// TIA Portal V16 export
// export: Created 2021-04-12T08:07:25.9683963Z, ExportSetting WithDefaults, DisplayName Totally Integrated Automation Portal, DisplayVersion V16, DisplayName TIA Portal Version Control Interface, DisplayVersion V16, DisplayName TIA Portal Openness, DisplayVersion V16, DisplayName STEP 7 Professional, DisplayVersion V16, DisplayName STEP 7 Safety, DisplayVersion V16, DisplayName WinCC Unified SCADA Engineering System, DisplayVersion V16
FUNCTION_BLOCK "AutoMode"   // FB20, LAD
TITLE = Автоматический режим
{ S7_Optimized_Access := 'TRUE' }
VERSION : 0.1
// //setWeight - уставка веса в упаковке => используется при подсчете уставок в бункера
// //speed_inConveyer - уставка скорости на питателе в %
// //speedVibro - уставка скорости вибрации в %
// //maxWeightBunker - максимальный вес в один бункер => используется при подсчете уставок в бункера
// //workPlavnik - использовать ли плавник во время работы 
// //measurementError - допустимая погрешность на итоговый вес => используется при поиске подходящих бункеров при сбросе
// //mediumWeightProduct - средний вес продукта => используется при подсчете уставок в бункера
// stored: AutoNumber false, IsIECCheckEnabled false, IsRetainMemResEnabled false, MemoryReserve 100, SetENOAutomatically false, UDAEnableTagReadback false
   VAR_IN_OUT
      enableAutoMode : Bool;   // разрешение на переход в автоматический режим
      isFinishPreWork : Bool;   // сигнал об окончании подготовки к автоматическому режиму
      isStartAutoMode : Bool;   // сигнал что автоматический режим запущен
   END_VAR
   VAR
      TaskSetWeight : Real;   // целевой вес который ищем в сортировке
      SetWeightBunker : Array[0..12] of Real;   // уставки весов в бункера
      currentWeightBunker : Array[0..12] of Real;
      readyToSort : Array[0..12] of Bool;   // массив говорящий какие бункера готовы к сортировке
      readyToDrop : Array[0..12] of Bool;   // массив говорящий какие бункера надо сбросить
      readyToDropYP : Array[0..2] of Bool;
      isWorkWithBunker : Array[0..12] of Bool;   // массив разрешающий бункерам работать
      preWorkAutoMode : Struct
         isFinishPreWork : Bool;
         alarmStop : Bool;
      END_STRUCT;
      preWork_AM_FB : "preWork_AM";
      workPackingMachine_AM_FB : "workPackingMachine_AM";
      workInConveyer_AM_FB : "workInConveyer_AM";
      controlFllipper_AM_FB : "controlValve";
      workVibroLot_AM_FB : Array[0..12] of "workVibroLot_AM";
      workVibroTable_AM_FB : "workVibroTable_AM";
      weightModule_AM_FB : "weightModule_AM";
      Sorting_AM_FB : "Sorting_AM";
      setWeightBunker_FB : "setWeightBunker_AM";
      blockSorting : Bool;   // запрет на сортировку в блоке сортировке
      openFlipper : Bool;
      hmiYpDropWeight : Array[0..2] of Real;
      hmiYpDropError : Array[0..2] of Real;
      Sorting_AM_withBuffer_FB { S7_SetPoint := 'True'} : "Sorting_AM_withBuffer";
   END_VAR
   VAR_TEMP
      "!!!!!" : Array[0..1] of Bool;
      i : DInt;
      tmpStableWeightBunker : Array[0..12] of Real;
   END_VAR
BEGIN

REGION Network 1: Аварийный останов
   // По нажатию кнопки Стоп и Аварийный стоп
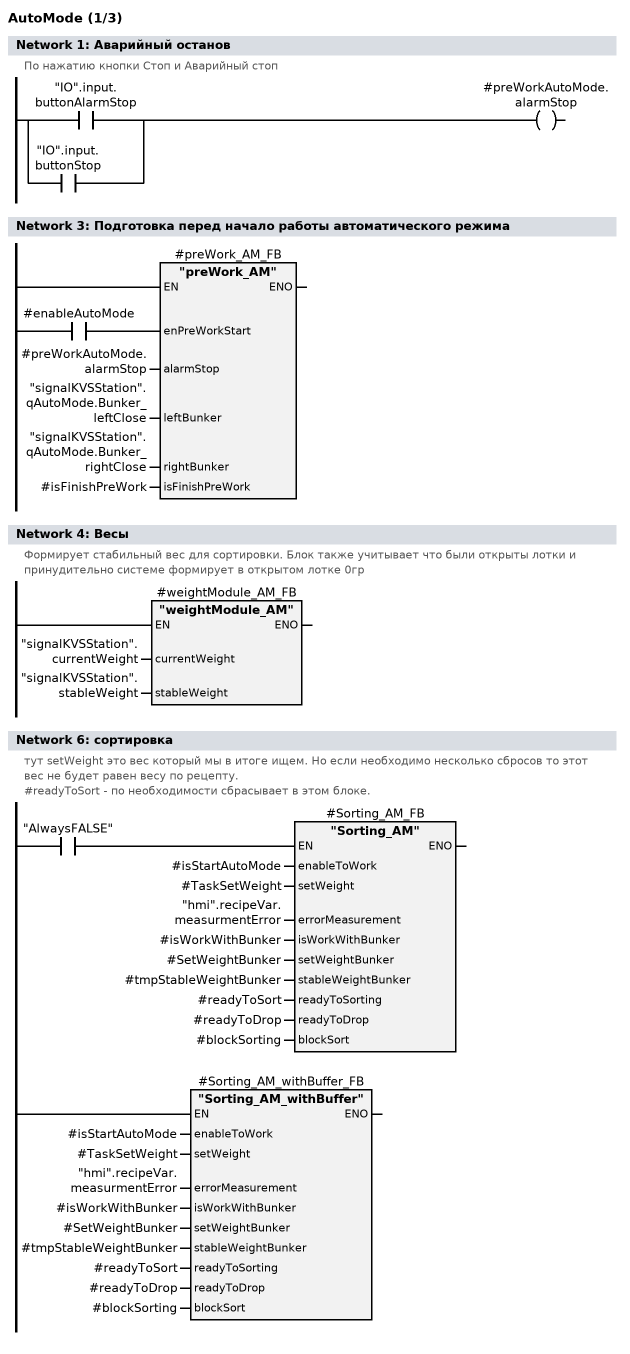
   RUNG wire#powerrail
      Contact( "IO".input.buttonAlarmStop )
      wire#w1
      Coil( #preWorkAutoMode.alarmStop )
   END_RUNG
   RUNG wire#powerrail
      Contact( "IO".input.buttonStop )
   END_RUNG wire#w1
   // the same network as SCL:
   #preWorkAutoMode.alarmStop := "IO".input.buttonAlarmStop OR "IO".input.buttonStop;
END_REGION

REGION Network 2 (SCL): статусы автоматического режима
   IF #enableAutoMode THEN
       IF NOT (#isFinishPreWork) THEN
           "hmi".readySystem := 2;
       ELSE
           IF NOT (#isStartAutoMode) THEN
               "hmi".readySystem := 0;
           ELSE
               "hmi".readySystem := 1;
           END_IF;
       END_IF;
   END_IF;
END_REGION

REGION Network 3: Подготовка перед начало работы автоматического режима
   RUNG wire#powerrail
      #preWork_AM_FB(enPreWorkStart := wire#w1, alarmStop := #preWorkAutoMode.alarmStop, leftBunker := "signalKVSStation".qAutoMode.Bunker_leftClose, rightBunker := "signalKVSStation".qAutoMode.Bunker_rightClose, isFinishPreWork := #isFinishPreWork)
   END_RUNG
   RUNG wire#powerrail
      Contact( #enableAutoMode )
   END_RUNG wire#w1
   // the same network as SCL:
   #preWork_AM_FB(enPreWorkStart := #enableAutoMode,   // "preWork_AM"
                  alarmStop := #preWorkAutoMode.alarmStop,
                  leftBunker := "signalKVSStation".qAutoMode.Bunker_leftClose,
                  rightBunker := "signalKVSStation".qAutoMode.Bunker_rightClose,
                  isFinishPreWork := #isFinishPreWork);
END_REGION

REGION Network 4: Весы
   // Формирует стабильный вес для сортировки. Блок также учитывает что были открыты лотки и принудительно системе формирует в открытом лотке 0гр
   RUNG wire#powerrail
      #weightModule_AM_FB(currentWeight := "signalKVSStation".currentWeight, stableWeight := "signalKVSStation".stableWeight)
   END_RUNG
   // the same network as SCL:
   #weightModule_AM_FB(currentWeight := "signalKVSStation".currentWeight,   // "weightModule_AM"
                       stableWeight := "signalKVSStation".stableWeight);
END_REGION

REGION Network 5 (SCL): выделяем стабильные веса с которыми будем работать
   #i := 0;
   FOR #i := 1 TO 12 DO
       #tmpStableWeightBunker[#i] := "signalKVSStation".stableWeight[#i].weight[0];
       "hmi".weightLine[#i].currentWeightPocket := "signalKVSStation".stableWeight[#i].weight[0];
       "hmi".weightLine[#i].targetWeightPocket := #SetWeightBunker[#i];
   END_FOR;
   #currentWeightBunker := "signalKVSStation".currentWeight;
END_REGION

REGION Network 6: сортировка
   // тут setWeight это вес который мы в итоге ищем. Но если необходимо несколько сбросов то этот вес не будет равен весу по рецепту.
   // #readyToSort - по необходимости сбрасывает в этом блоке.
   RUNG wire#powerrail
      Contact( "AlwaysFALSE" )
      #Sorting_AM_FB(enableToWork := #isStartAutoMode, setWeight := #TaskSetWeight, errorMeasurement := "hmi".recipeVar.measurmentError, isWorkWithBunker := #isWorkWithBunker, setWeightBunker := #SetWeightBunker, stableWeightBunker := #tmpStableWeightBunker, readyToSorting := #readyToSort, readyToDrop := #readyToDrop, blockSort := #blockSorting)
   END_RUNG
   RUNG wire#powerrail
      #Sorting_AM_withBuffer_FB(enableToWork := #isStartAutoMode, setWeight := #TaskSetWeight, errorMeasurement := "hmi".recipeVar.measurmentError, isWorkWithBunker := #isWorkWithBunker, setWeightBunker := #SetWeightBunker, stableWeightBunker := #tmpStableWeightBunker, readyToSorting := #readyToSort, readyToDrop := #readyToDrop, blockSort := #blockSorting)
   END_RUNG
   // the same network as SCL:
   IF "AlwaysFALSE" THEN
       #Sorting_AM_FB(enableToWork := #isStartAutoMode,   // "Sorting_AM"
                      setWeight := #TaskSetWeight,
                      errorMeasurement := "hmi".recipeVar.measurmentError,
                      isWorkWithBunker := #isWorkWithBunker,
                      setWeightBunker := #SetWeightBunker,
                      stableWeightBunker := #tmpStableWeightBunker,
                      readyToSorting := #readyToSort,
                      readyToDrop := #readyToDrop,
                      blockSort := #blockSorting);
   END_IF;
   #Sorting_AM_withBuffer_FB(enableToWork := #isStartAutoMode,   // "Sorting_AM_withBuffer"
                           setWeight := #TaskSetWeight,
                           errorMeasurement := "hmi".recipeVar.measurmentError,
                           isWorkWithBunker := #isWorkWithBunker,
                           setWeightBunker := #SetWeightBunker,
                           stableWeightBunker := #tmpStableWeightBunker,
                           readyToSorting := #readyToSort,
                           readyToDrop := #readyToDrop,
                           blockSort := #blockSorting);
END_REGION

REGION Network 7 (SCL): Перенос данных для панели
   "hmi".permitOn1Bunk := "hmi".permitOn2Bunk := #readyToDrop;
END_REGION

REGION Network 8: Расчет уставок в бункере
   // Здесь происходит расчет уставок на все бункера в зависимости от: веса уставки, максимального веса в один бункер, среднего веса продукта
   // Также управление конвейерами, упаковочными машинами и бункерами
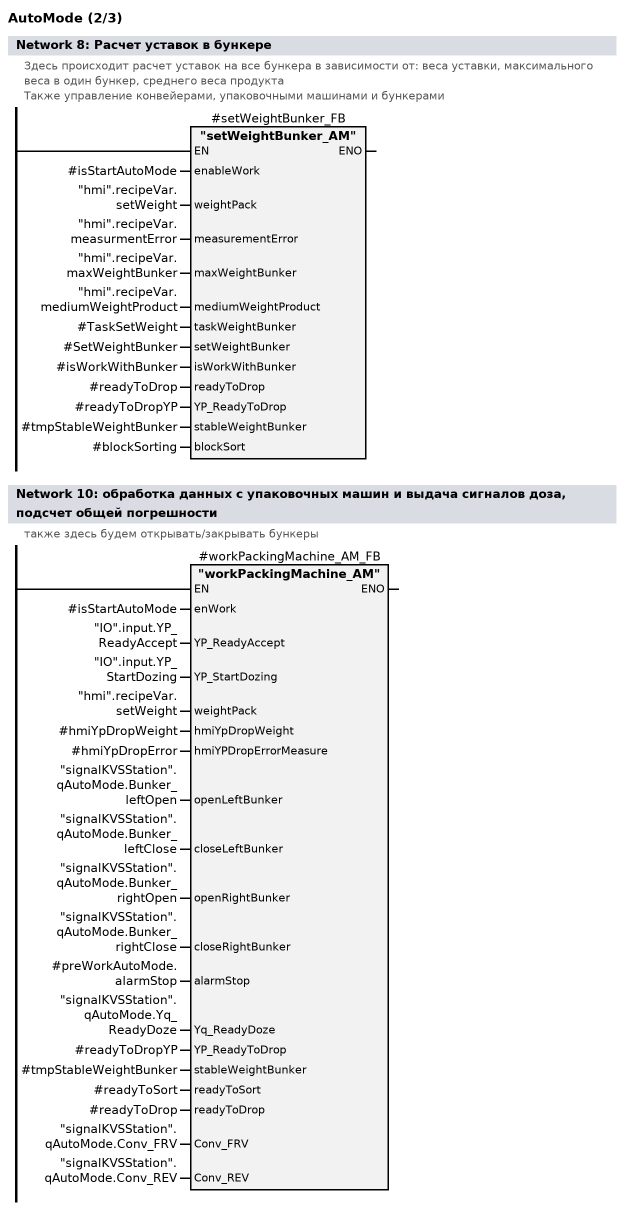
   RUNG wire#powerrail
      #setWeightBunker_FB(enableWork := #isStartAutoMode, weightPack := "hmi".recipeVar.setWeight, measurementError := "hmi".recipeVar.measurmentError, maxWeightBunker := "hmi".recipeVar.maxWeightBunker, mediumWeightProduct := "hmi".recipeVar.mediumWeightProduct, taskWeightBunker := #TaskSetWeight, setWeightBunker := #SetWeightBunker, isWorkWithBunker := #isWorkWithBunker, readyToDrop := #readyToDrop, YP_ReadyToDrop := #readyToDropYP, stableWeightBunker := #tmpStableWeightBunker, blockSort := #blockSorting)
   END_RUNG
   // the same network as SCL:
   #setWeightBunker_FB(enableWork := #isStartAutoMode,   // "setWeightBunker_AM"
                       weightPack := "hmi".recipeVar.setWeight,
                       measurementError := "hmi".recipeVar.measurmentError,
                       maxWeightBunker := "hmi".recipeVar.maxWeightBunker,
                       mediumWeightProduct := "hmi".recipeVar.mediumWeightProduct,
                       taskWeightBunker := #TaskSetWeight,
                       setWeightBunker := #SetWeightBunker,
                       isWorkWithBunker := #isWorkWithBunker,
                       readyToDrop := #readyToDrop,
                       YP_ReadyToDrop := #readyToDropYP,
                       stableWeightBunker := #tmpStableWeightBunker,
                       blockSort := #blockSorting);
END_REGION

REGION Network 9 (SCL): передача уставок в панель
   #i := 0;
   FOR #i := 1 TO 12 DO
       "hmi".weightLine[#i].targetWeightPocket := #SetWeightBunker[#i];
   END_FOR;
END_REGION

REGION Network 10: обработка данных с упаковочных машин и выдача сигналов доза, подсчет общей погрешности
   // также здесь будем открывать/закрывать бункеры
   RUNG wire#powerrail
      #workPackingMachine_AM_FB(enWork := #isStartAutoMode, YP_ReadyAccept := "IO".input.YP_ReadyAccept, YP_StartDozing := "IO".input.YP_StartDozing, weightPack := "hmi".recipeVar.setWeight, hmiYpDropWeight := #hmiYpDropWeight, hmiYPDropErrorMeasure := #hmiYpDropError, openLeftBunker := "signalKVSStation".qAutoMode.Bunker_leftOpen, closeLeftBunker := "signalKVSStation".qAutoMode.Bunker_leftClose, openRightBunker := "signalKVSStation".qAutoMode.Bunker_rightOpen, closeRightBunker := "signalKVSStation".qAutoMode.Bunker_rightClose, alarmStop := #preWorkAutoMode.alarmStop, Yq_ReadyDoze := "signalKVSStation".qAutoMode.Yq_ReadyDoze, YP_ReadyToDrop := #readyToDropYP, stableWeightBunker := #tmpStableWeightBunker, readyToSort := #readyToSort, readyToDrop := #readyToDrop, Conv_FRV := "signalKVSStation".qAutoMode.Conv_FRV, Conv_REV := "signalKVSStation".qAutoMode.Conv_REV)
   END_RUNG
   // the same network as SCL:
   #workPackingMachine_AM_FB(enWork := #isStartAutoMode,   // "workPackingMachine_AM"
                           YP_ReadyAccept := "IO".input.YP_ReadyAccept,
                           YP_StartDozing := "IO".input.YP_StartDozing,
                           weightPack := "hmi".recipeVar.setWeight,
                           hmiYpDropWeight := #hmiYpDropWeight,
                           hmiYPDropErrorMeasure := #hmiYpDropError,
                           openLeftBunker := "signalKVSStation".qAutoMode.Bunker_leftOpen,
                           closeLeftBunker := "signalKVSStation".qAutoMode.Bunker_leftClose,
                           openRightBunker := "signalKVSStation".qAutoMode.Bunker_rightOpen,
                           closeRightBunker := "signalKVSStation".qAutoMode.Bunker_rightClose,
                           alarmStop := #preWorkAutoMode.alarmStop,
                           Yq_ReadyDoze := "signalKVSStation".qAutoMode.Yq_ReadyDoze,
                           YP_ReadyToDrop := #readyToDropYP,
                           stableWeightBunker := #tmpStableWeightBunker,
                           readyToSort := #readyToSort,
                           readyToDrop := #readyToDrop,
                           Conv_FRV := "signalKVSStation".qAutoMode.Conv_FRV,
                           Conv_REV := "signalKVSStation".qAutoMode.Conv_REV);
END_REGION

REGION Network 11 (SCL)
   #i := 0;
   FOR #i := 1 TO 2 DO
       "hmi".outConvAndPack[#i].currentWeightPack := #hmiYpDropWeight[#i];
       "hmi".outConvAndPack[#i].currentErrorMeasure := #hmiYpDropError[#i];
   END_FOR;
END_REGION

REGION Network 12: Работа конвейера
   // конвейер работает пока не сработал датчик пересыпа
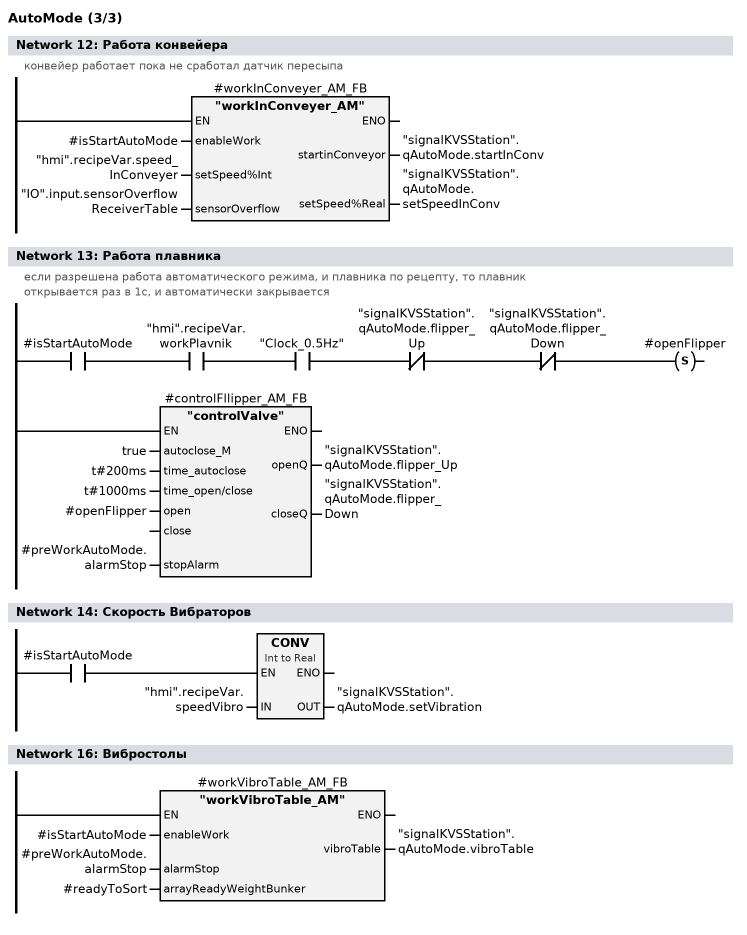
   RUNG wire#powerrail
      #workInConveyer_AM_FB(enableWork := #isStartAutoMode, "setSpeed%Int" := "hmi".recipeVar.speed_InConveyer, sensorOverflow := "IO".input.sensorOverflowReceiverTable, startinConveyor => "signalKVSStation".qAutoMode.startInConv, "setSpeed%Real" => "signalKVSStation".qAutoMode.setSpeedInConv)
   END_RUNG
   // the same network as SCL:
   #workInConveyer_AM_FB(enableWork := #isStartAutoMode,   // "workInConveyer_AM"
                         "setSpeed%Int" := "hmi".recipeVar.speed_InConveyer,
                         sensorOverflow := "IO".input.sensorOverflowReceiverTable,
                         startinConveyor => "signalKVSStation".qAutoMode.startInConv,
                         "setSpeed%Real" => "signalKVSStation".qAutoMode.setSpeedInConv);
END_REGION

REGION Network 13: Работа плавника
   // если разрешена работа автоматического режима, и плавника по рецепту, то плавник
   // открывается раз в 1с, и автоматически закрывается
   RUNG wire#powerrail
      Contact( #isStartAutoMode )
      Contact( "hmi".recipeVar.workPlavnik )
      Contact( "Clock_0.5Hz" )
      I_Contact( "signalKVSStation".qAutoMode.flipper_Up )
      I_Contact( "signalKVSStation".qAutoMode.flipper_Down )
      S_Coil( #openFlipper )
   END_RUNG
   RUNG wire#powerrail
      #controlFllipper_AM_FB(autoclose_M := true, time_autoclose := t#200ms, "time_open/close" := t#1000ms, open := #openFlipper, close :=, stopAlarm := #preWorkAutoMode.alarmStop, openQ => "signalKVSStation".qAutoMode.flipper_Up, closeQ => "signalKVSStation".qAutoMode.flipper_Down)
   END_RUNG
   // the same network as SCL:
   IF #isStartAutoMode AND "hmi".recipeVar.workPlavnik AND "Clock_0.5Hz" AND NOT "signalKVSStation".qAutoMode.flipper_Up AND NOT "signalKVSStation".qAutoMode.flipper_Down THEN
       #openFlipper := TRUE;
   END_IF;
   #controlFllipper_AM_FB(autoclose_M := true,   // "controlValve"
                          time_autoclose := t#200ms,
                          "time_open/close" := t#1000ms,
                          open := #openFlipper,
                          stopAlarm := #preWorkAutoMode.alarmStop,
                          openQ => "signalKVSStation".qAutoMode.flipper_Up,
                          closeQ => "signalKVSStation".qAutoMode.flipper_Down);
END_REGION

REGION Network 14: Скорость Вибраторов
   RUNG wire#powerrail
      Contact( #isStartAutoMode )
      { S7_Templates := "[SrcType := Int, DestType := Real]" } Convert(in := "hmi".recipeVar.speedVibro, out => "signalKVSStation".qAutoMode.setVibration)
   END_RUNG
   // the same network as SCL:
   IF #isStartAutoMode THEN
       "signalKVSStation".qAutoMode.setVibration := INT_TO_REAL("hmi".recipeVar.speedVibro);
   END_IF;
END_REGION

REGION Network 15 (SCL): Вибролотки, лопатки
   #i := 0;
   FOR #i := 1 TO 12 DO
       #workVibroLot_AM_FB[#i](enableWork := #isStartAutoMode,
                               setWeightBunker := #SetWeightBunker[#i],
                               currentWeight := #currentWeightBunker[#i],//"signalKVSStation".stableWeight[#i].weight[0],
                               stateDoor := "hmi".weightLine[#i].stateValveAfterVibroLot,
                               stateBunkerLeft:="hmi".weightLine[#i].stateLeftValveWeightPocket,
                               stateBunkerRight:="hmi".weightLine[#i].stateRightValveWeightPocket,
                               alarmStop := #preWorkAutoMode.alarmStop,
                               isWorkWithBunker := #isWorkWithBunker[#i],

                               onVibroLot:= "signalKVSStation".qAutoMode.vibroLot[#i],
                               openDoor := "signalKVSStation".qAutoMode.Door_open[#i],
                               closeDoor := "signalKVSStation".qAutoMode.Door_close[#i],

                               isReadyToDrop:=#readyToDrop[#i],
                               isReadyToSort := #readyToSort[#i]);

   END_FOR;
END_REGION

REGION Network 16: Вибростолы
   RUNG wire#powerrail
      #workVibroTable_AM_FB(enableWork := #isStartAutoMode, alarmStop := #preWorkAutoMode.alarmStop, arrayReadyWeightBunker := #readyToSort, vibroTable => "signalKVSStation".qAutoMode.vibroTable)
   END_RUNG
   // the same network as SCL:
   #workVibroTable_AM_FB(enableWork := #isStartAutoMode,   // "workVibroTable_AM"
                         alarmStop := #preWorkAutoMode.alarmStop,
                         arrayReadyWeightBunker := #readyToSort,
                         vibroTable => "signalKVSStation".qAutoMode.vibroTable);
END_REGION
END_FUNCTION_BLOCK
